{attribute addProperty BoxType "EK1100-0000-0018"}
{attribute addProperty Id "A_0014_BK1250_0000_0000A_0014_BK1250_0000_0000_A4796D4900"}
{attribute addProperty CRC "3458156838"}
{attribute addProperty SizeInBites "0"}
{attribute addProperty SizeInBytes "0"}
TYPE Beckhoff_BKxxxxsub_EK1100_CE1F4926 EXTENDS EK1100_179A0949 :
STRUCT
	{attribute addProperty Name "A_0014_BK1250_0000_0000"}
	A_0014_BK1250_0000_0000 : A_0014_BK1250_0000_0000_A4796D49;
END_STRUCT
END_TYPE

(* stored: Version 1.2.0.0, ProductVersion 3.1.4024.9
   DUT Beckhoff_BKxxxxsub_EK1100_CE1F4926: Id {a9f9f0d6-2d01-4875-b180-447276a635f9} *)
